// TIA Portal V16 export
// export: Created 2022-02-04T14:40:20.664957Z, ExportSetting WithDefaults, DisplayName Totally Integrated Automation Portal, DisplayVersion V16 Update 1, DisplayName TIA Portal Version Control Interface, DisplayVersion V16, DisplayName TIA Portal Openness, DisplayVersion V16, DisplayName SINAMICS Startdrive Advanced, DisplayVersion V16 Update 5, DisplayName SINAMICS Startdrive G130, G150, S120, S150, SINAMICS MV, S210, DisplayVersion V16 Update 5, DisplayName SINAMICS Startdrive G110M, G120, G120C, G120D, G120P, G115D, DisplayVersion V16 Update 5, DisplayName STEP 7 Professional, DisplayVersion V16, DisplayName STEP 7 Safety, DisplayVersion V16, DisplayName WinCC Advanced, DisplayVersion V16, DisplayName SIMATIC Visualization Architect, DisplayVersion V16
DATA_BLOCK "UporPFM_DB"   // DB12
VERSION : 0.1
// stored: AutoNumber true, InstanceOfName UporPFM, InstanceOfType FB
"UporPFM"
   // VAR_INPUT
   //    firstWheel : Bool;
   //    secondWheel : Bool;
   //    boardSensorClose : Bool;
   //    boardSensorFar : Bool;
   //    readyStartPacket : Bool;
   //    stopTask : Bool;
   //    NoChessLayout : Bool;
   //    MuchBoards : Bool;
   //    ResetFaults : Bool;
   //    Correcting : Bool;
   //    CorrectCounters : Bool;
   //    CorrectedWheel : Bool;
   //    BoardsInLay : Int;
   //    Length : Int;
   //    CorrectedCounter : Int;
   // END_VAR
   // VAR_OUTPUT
   //    CMD_Up : Bool;
   //    CMD_Down : Bool;
   //    CommonAlarm : Bool;
   //    AlarmGidra : Bool;
   //    AlarmWarpingBoard : Bool;
   // END_VAR
   // VAR RETAIN
   //    firstWheel_old : Bool;
   //    secondWheel_old : Bool;
   //    muchBoards_old : Bool;
   //    boardSensor_old : Bool;
   //    currentSelectedWheel : Bool;
   //    needWork : Bool;
   //    haveTask : Bool;
   //    Skip : Bool;
   //    DenyAlarm : Bool;
   //    helper : Bool;
   //    "Counter" : Int;
   //    notAwaitableBoard_timer : TON;
   //    notStableLayer_timer { S7_SetPoint := 'True'} : TOF;
   //    StableLayer_timer { S7_SetPoint := 'True'} : TON;
   // END_VAR
BEGIN
END_DATA_BLOCK
